PROGRAM PRG_COM
VAR
END_VAR

(*Instanitate Serial port com function *) 
	
fbSerialLineControl_CVMI_ROUGH_PTM_01(
	Mode:= SERIALLINEMODE_EL6_22B,
	pComIn:= ADR(stComIn_CVMI_ROUGH_PTM_01),
	pComOut:=ADR(stComOut_CVMI_ROUGH_PTM_01),
	SizeComIn:= SIZEOF(stComIn_CVMI_ROUGH_PTM_01),
	TxBuffer:= SerialTXBuffer_CVMI_ROUGH_PTM_01,
	RxBuffer:= SerialRXBuffer_CVMI_ROUGH_PTM_01,
	Error=> ,
	ErrorID=> );
	
fbSerialLineControl_CVMI_KTOF_PTM_01(
	Mode:= SERIALLINEMODE_EL6_22B,
	pComIn:= ADR(stComIn_CVMI_KTOF_PTM_01),
	pComOut:=ADR(stComOut_CVMI_KTOF_PTM_01),
	SizeComIn:= SIZEOF(stComIn_CVMI_KTOF_PTM_01),
	TxBuffer:= SerialTXBuffer_CVMI_KTOF_PTM_01,
	RxBuffer:= SerialRXBuffer_CVMI_KTOF_PTM_01,
	Error=> ,
	ErrorID=> );
	
fbSerialLineControl_CVMI_KTOF_PTM_02(
	Mode:= SERIALLINEMODE_EL6_22B,
	pComIn:= ADR(stComIn_CVMI_KTOF_PTM_02),
	pComOut:=ADR(stComOut_CVMI_KTOF_PTM_02),
	SizeComIn:= SIZEOF(stComIn_CVMI_KTOF_PTM_02),
	TxBuffer:= SerialTXBuffer_CVMI_KTOF_PTM_02,
	RxBuffer:= SerialRXBuffer_CVMI_KTOF_PTM_02,
	Error=> ,
	ErrorID=> );

END_PROGRAM

(* stored: Version 1.1.0.1, ProductVersion 3.1.4024.6
   POU PRG_COM: Id {cd596418-8e0a-453c-867e-618b97030684}, SpecialFunc None *)
